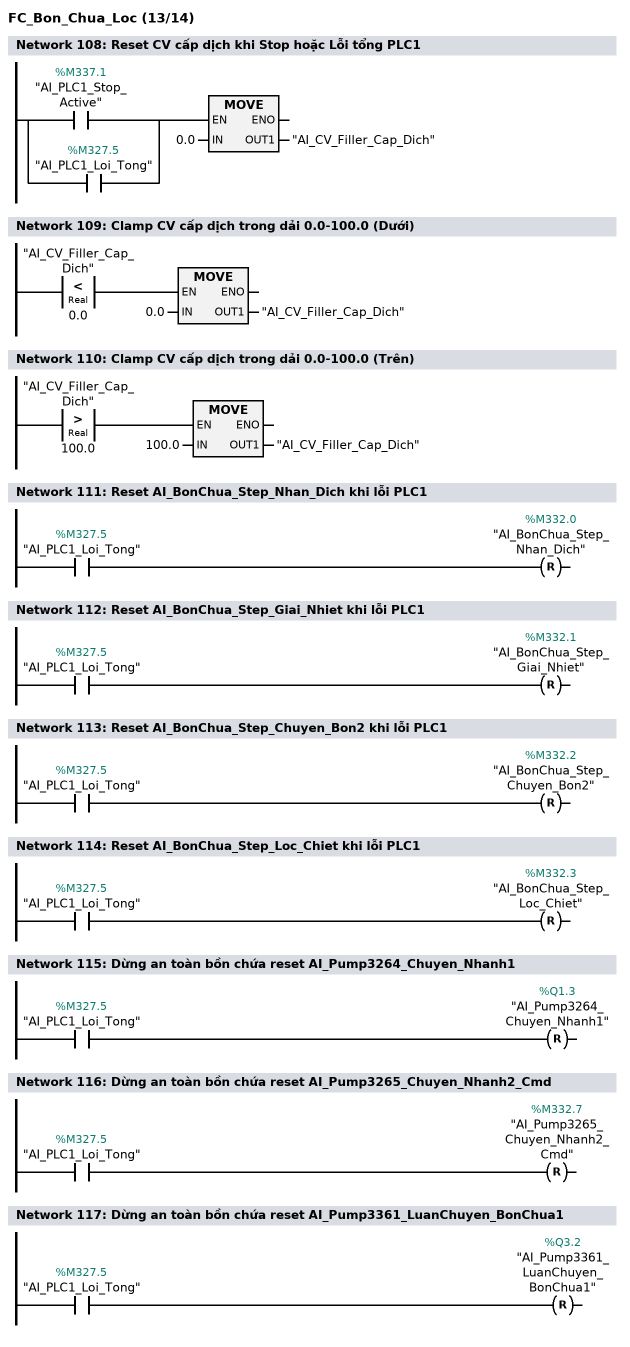
   RUNG wire#powerrail
      Contact( "AI_PLC1_Stop_Active" )
      wire#w1
      { S7_GenerateENO := "TRUE" } Move(in := 0.0, out1 => "AI_CV_Filler_Cap_Dich")
   END_RUNG
   RUNG wire#powerrail
      Contact( "AI_PLC1_Loi_Tong" )
   END_RUNG wire#w1
   // the same network as SCL:
   IF "AI_PLC1_Stop_Active" OR "AI_PLC1_Loi_Tong" THEN "AI_CV_Filler_Cap_Dich" := 0.0; END_IF;
END_REGION

REGION Network 109: Clamp CV cấp dịch trong dải 0.0-100.0 (Dưới)
   RUNG wire#powerrail
      { S7_Templates := "SrcType := Real" } LT_Contact(in1 := "AI_CV_Filler_Cap_Dich", in2 := 0.0)
      { S7_GenerateENO := "TRUE" } Move(in := 0.0, out1 => "AI_CV_Filler_Cap_Dich")
   END_RUNG
   // the same network as SCL:
   IF "AI_CV_Filler_Cap_Dich" < 0.0 THEN "AI_CV_Filler_Cap_Dich" := 0.0; END_IF;
END_REGION

REGION Network 110: Clamp CV cấp dịch trong dải 0.0-100.0 (Trên)
   RUNG wire#powerrail
      { S7_Templates := "SrcType := Real" } GT_Contact(in1 := "AI_CV_Filler_Cap_Dich", in2 := 100.0)
      { S7_GenerateENO := "TRUE" } Move(in := 100.0, out1 => "AI_CV_Filler_Cap_Dich")
   END_RUNG
   // the same network as SCL:
   IF "AI_CV_Filler_Cap_Dich" > 100.0 THEN "AI_CV_Filler_Cap_Dich" := 100.0; END_IF;
END_REGION

REGION Network 111: Reset AI_BonChua_Step_Nhan_Dich khi lỗi PLC1
   RUNG wire#powerrail
      Contact( "AI_PLC1_Loi_Tong" )
      R_Coil( "AI_BonChua_Step_Nhan_Dich" )
   END_RUNG
   // the same network as SCL:
   IF "AI_PLC1_Loi_Tong" THEN "AI_BonChua_Step_Nhan_Dich" := FALSE; END_IF;
END_REGION

REGION Network 112: Reset AI_BonChua_Step_Giai_Nhiet khi lỗi PLC1
   RUNG wire#powerrail
      Contact( "AI_PLC1_Loi_Tong" )
      R_Coil( "AI_BonChua_Step_Giai_Nhiet" )
   END_RUNG
   // the same network as SCL:
   IF "AI_PLC1_Loi_Tong" THEN "AI_BonChua_Step_Giai_Nhiet" := FALSE; END_IF;
END_REGION

REGION Network 113: Reset AI_BonChua_Step_Chuyen_Bon2 khi lỗi PLC1
   RUNG wire#powerrail
      Contact( "AI_PLC1_Loi_Tong" )
      R_Coil( "AI_BonChua_Step_Chuyen_Bon2" )
   END_RUNG
   // the same network as SCL:
   IF "AI_PLC1_Loi_Tong" THEN "AI_BonChua_Step_Chuyen_Bon2" := FALSE; END_IF;
END_REGION

REGION Network 114: Reset AI_BonChua_Step_Loc_Chiet khi lỗi PLC1
   RUNG wire#powerrail
      Contact( "AI_PLC1_Loi_Tong" )
      R_Coil( "AI_BonChua_Step_Loc_Chiet" )
   END_RUNG
   // the same network as SCL:
   IF "AI_PLC1_Loi_Tong" THEN "AI_BonChua_Step_Loc_Chiet" := FALSE; END_IF;
END_REGION

REGION Network 115: Dừng an toàn bồn chứa reset AI_Pump3264_Chuyen_Nhanh1
   RUNG wire#powerrail
      Contact( "AI_PLC1_Loi_Tong" )
      R_Coil( "AI_Pump3264_Chuyen_Nhanh1" )
   END_RUNG
   // the same network as SCL:
   IF "AI_PLC1_Loi_Tong" THEN "AI_Pump3264_Chuyen_Nhanh1" := FALSE; END_IF;
END_REGION

REGION Network 116: Dừng an toàn bồn chứa reset AI_Pump3265_Chuyen_Nhanh2_Cmd
   RUNG wire#powerrail
      Contact( "AI_PLC1_Loi_Tong" )
      R_Coil( "AI_Pump3265_Chuyen_Nhanh2_Cmd" )
   END_RUNG
   // the same network as SCL:
   IF "AI_PLC1_Loi_Tong" THEN "AI_Pump3265_Chuyen_Nhanh2_Cmd" := FALSE; END_IF;
END_REGION

REGION Network 117: Dừng an toàn bồn chứa reset AI_Pump3361_LuanChuyen_BonChua1
   RUNG wire#powerrail
      Contact( "AI_PLC1_Loi_Tong" )
      R_Coil( "AI_Pump3361_LuanChuyen_BonChua1" )
   END_RUNG
   // the same network as SCL:
   IF "AI_PLC1_Loi_Tong" THEN "AI_Pump3361_LuanChuyen_BonChua1" := FALSE; END_IF;
END_REGION

REGION Network 118: Dừng an toàn bồn chứa reset AI_Pump3362_Xa_BonChua1
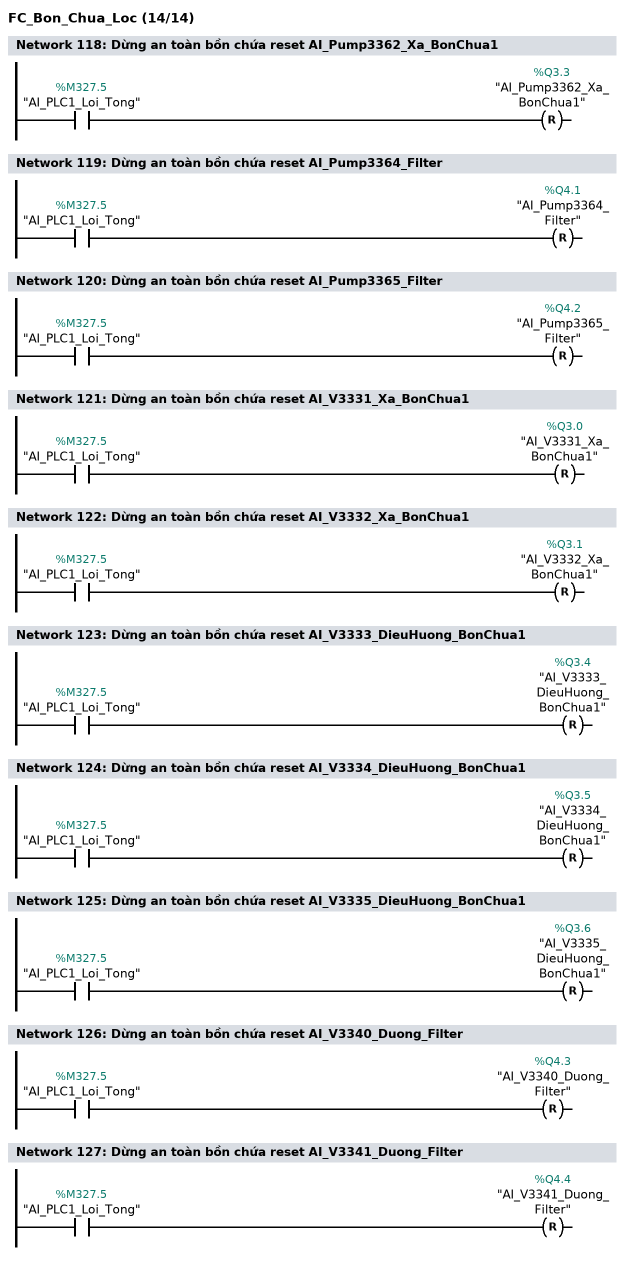
   RUNG wire#powerrail
      Contact( "AI_PLC1_Loi_Tong" )
      R_Coil( "AI_Pump3362_Xa_BonChua1" )
   END_RUNG
   // the same network as SCL:
   IF "AI_PLC1_Loi_Tong" THEN "AI_Pump3362_Xa_BonChua1" := FALSE; END_IF;
END_REGION

REGION Network 119: Dừng an toàn bồn chứa reset AI_Pump3364_Filter
   RUNG wire#powerrail
      Contact( "AI_PLC1_Loi_Tong" )
      R_Coil( "AI_Pump3364_Filter" )
   END_RUNG
   // the same network as SCL:
   IF "AI_PLC1_Loi_Tong" THEN "AI_Pump3364_Filter" := FALSE; END_IF;
END_REGION

REGION Network 120: Dừng an toàn bồn chứa reset AI_Pump3365_Filter
   RUNG wire#powerrail
      Contact( "AI_PLC1_Loi_Tong" )
      R_Coil( "AI_Pump3365_Filter" )
   END_RUNG
   // the same network as SCL:
   IF "AI_PLC1_Loi_Tong" THEN "AI_Pump3365_Filter" := FALSE; END_IF;
END_REGION

REGION Network 121: Dừng an toàn bồn chứa reset AI_V3331_Xa_BonChua1
   RUNG wire#powerrail
      Contact( "AI_PLC1_Loi_Tong" )
      R_Coil( "AI_V3331_Xa_BonChua1" )
   END_RUNG
   // the same network as SCL:
   IF "AI_PLC1_Loi_Tong" THEN "AI_V3331_Xa_BonChua1" := FALSE; END_IF;
END_REGION

REGION Network 122: Dừng an toàn bồn chứa reset AI_V3332_Xa_BonChua1
   RUNG wire#powerrail
      Contact( "AI_PLC1_Loi_Tong" )
      R_Coil( "AI_V3332_Xa_BonChua1" )
   END_RUNG
   // the same network as SCL:
   IF "AI_PLC1_Loi_Tong" THEN "AI_V3332_Xa_BonChua1" := FALSE; END_IF;
END_REGION

REGION Network 123: Dừng an toàn bồn chứa reset AI_V3333_DieuHuong_BonChua1
   RUNG wire#powerrail
      Contact( "AI_PLC1_Loi_Tong" )
      R_Coil( "AI_V3333_DieuHuong_BonChua1" )
   END_RUNG
   // the same network as SCL:
   IF "AI_PLC1_Loi_Tong" THEN "AI_V3333_DieuHuong_BonChua1" := FALSE; END_IF;
END_REGION

REGION Network 124: Dừng an toàn bồn chứa reset AI_V3334_DieuHuong_BonChua1
   RUNG wire#powerrail
      Contact( "AI_PLC1_Loi_Tong" )
      R_Coil( "AI_V3334_DieuHuong_BonChua1" )
   END_RUNG
   // the same network as SCL:
   IF "AI_PLC1_Loi_Tong" THEN "AI_V3334_DieuHuong_BonChua1" := FALSE; END_IF;
END_REGION

REGION Network 125: Dừng an toàn bồn chứa reset AI_V3335_DieuHuong_BonChua1
   RUNG wire#powerrail
      Contact( "AI_PLC1_Loi_Tong" )
      R_Coil( "AI_V3335_DieuHuong_BonChua1" )
   END_RUNG
   // the same network as SCL:
   IF "AI_PLC1_Loi_Tong" THEN "AI_V3335_DieuHuong_BonChua1" := FALSE; END_IF;
END_REGION

REGION Network 126: Dừng an toàn bồn chứa reset AI_V3340_Duong_Filter
   RUNG wire#powerrail
      Contact( "AI_PLC1_Loi_Tong" )
      R_Coil( "AI_V3340_Duong_Filter" )
   END_RUNG
   // the same network as SCL:
   IF "AI_PLC1_Loi_Tong" THEN "AI_V3340_Duong_Filter" := FALSE; END_IF;
END_REGION

REGION Network 127: Dừng an toàn bồn chứa reset AI_V3341_Duong_Filter
   RUNG wire#powerrail
      Contact( "AI_PLC1_Loi_Tong" )
      R_Coil( "AI_V3341_Duong_Filter" )
   END_RUNG
   // the same network as SCL:
   IF "AI_PLC1_Loi_Tong" THEN "AI_V3341_Duong_Filter" := FALSE; END_IF;
END_REGION
END_FUNCTION

FUNCTION "FC_HMI_Mirror_PLC1" : Void   // FC40, LAD
{ S7_Optimized_Access := 'TRUE' }
VERSION : 0.1
// stored: AutoNumber true, IsIECCheckEnabled false, SetENOAutomatically false, UDAEnableTagReadback false
BEGIN

REGION Network 1: Mirror AI_V3230_Nuoc_Bon1
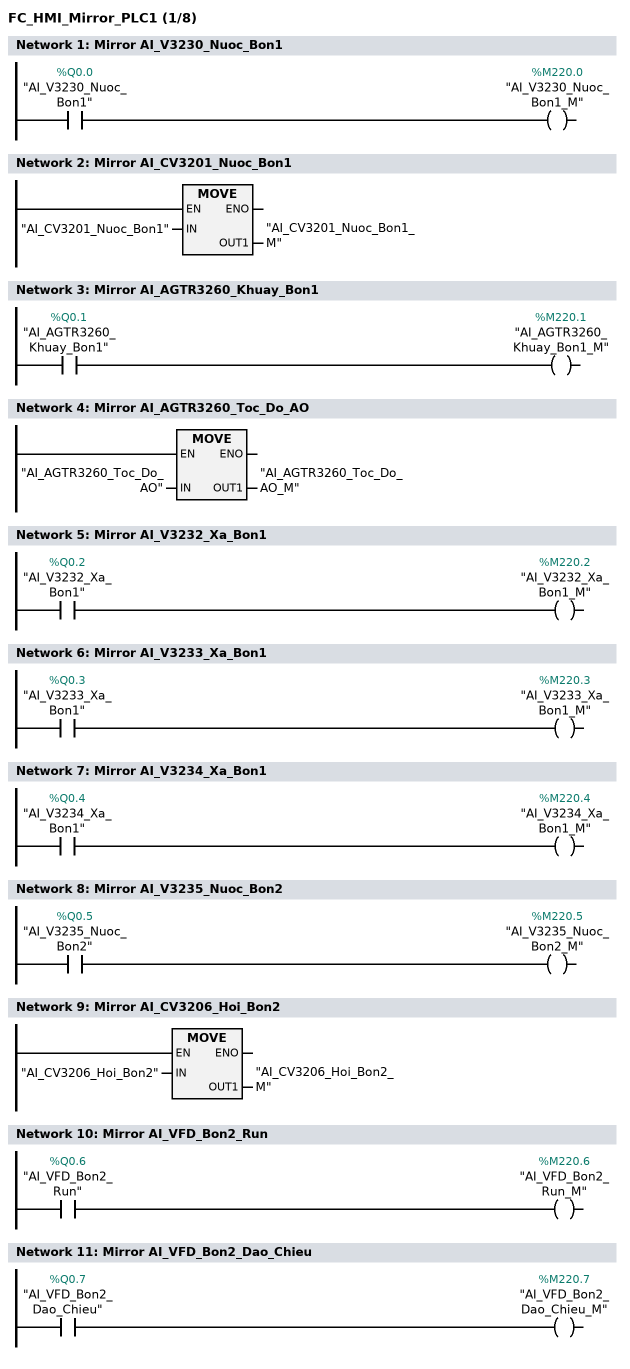
   RUNG wire#powerrail
      Contact( "AI_V3230_Nuoc_Bon1" )
      Coil( "AI_V3230_Nuoc_Bon1_M" )
   END_RUNG
   // the same network as SCL:
   "AI_V3230_Nuoc_Bon1_M" := "AI_V3230_Nuoc_Bon1";
END_REGION

REGION Network 2: Mirror AI_CV3201_Nuoc_Bon1
   RUNG wire#powerrail
      { S7_GenerateENO := "TRUE" } Move(in := "AI_CV3201_Nuoc_Bon1", out1 => "AI_CV3201_Nuoc_Bon1_M")
   END_RUNG
   // the same network as SCL:
   "AI_CV3201_Nuoc_Bon1_M" := "AI_CV3201_Nuoc_Bon1";
END_REGION

REGION Network 3: Mirror AI_AGTR3260_Khuay_Bon1
   RUNG wire#powerrail
      Contact( "AI_AGTR3260_Khuay_Bon1" )
      Coil( "AI_AGTR3260_Khuay_Bon1_M" )
   END_RUNG
   // the same network as SCL:
   "AI_AGTR3260_Khuay_Bon1_M" := "AI_AGTR3260_Khuay_Bon1";
END_REGION

REGION Network 4: Mirror AI_AGTR3260_Toc_Do_AO
   RUNG wire#powerrail
      { S7_GenerateENO := "TRUE" } Move(in := "AI_AGTR3260_Toc_Do_AO", out1 => "AI_AGTR3260_Toc_Do_AO_M")
   END_RUNG
   // the same network as SCL:
   "AI_AGTR3260_Toc_Do_AO_M" := "AI_AGTR3260_Toc_Do_AO";
END_REGION

REGION Network 5: Mirror AI_V3232_Xa_Bon1
   RUNG wire#powerrail
      Contact( "AI_V3232_Xa_Bon1" )
      Coil( "AI_V3232_Xa_Bon1_M" )
   END_RUNG
   // the same network as SCL:
   "AI_V3232_Xa_Bon1_M" := "AI_V3232_Xa_Bon1";
END_REGION

REGION Network 6: Mirror AI_V3233_Xa_Bon1
   RUNG wire#powerrail
      Contact( "AI_V3233_Xa_Bon1" )
      Coil( "AI_V3233_Xa_Bon1_M" )
   END_RUNG
   // the same network as SCL:
   "AI_V3233_Xa_Bon1_M" := "AI_V3233_Xa_Bon1";
END_REGION

REGION Network 7: Mirror AI_V3234_Xa_Bon1
   RUNG wire#powerrail
      Contact( "AI_V3234_Xa_Bon1" )
      Coil( "AI_V3234_Xa_Bon1_M" )
   END_RUNG
   // the same network as SCL:
   "AI_V3234_Xa_Bon1_M" := "AI_V3234_Xa_Bon1";
END_REGION

REGION Network 8: Mirror AI_V3235_Nuoc_Bon2
   RUNG wire#powerrail
      Contact( "AI_V3235_Nuoc_Bon2" )
      Coil( "AI_V3235_Nuoc_Bon2_M" )
   END_RUNG
   // the same network as SCL:
   "AI_V3235_Nuoc_Bon2_M" := "AI_V3235_Nuoc_Bon2";
END_REGION

REGION Network 9: Mirror AI_CV3206_Hoi_Bon2
   RUNG wire#powerrail
      { S7_GenerateENO := "TRUE" } Move(in := "AI_CV3206_Hoi_Bon2", out1 => "AI_CV3206_Hoi_Bon2_M")
   END_RUNG
   // the same network as SCL:
   "AI_CV3206_Hoi_Bon2_M" := "AI_CV3206_Hoi_Bon2";
END_REGION

REGION Network 10: Mirror AI_VFD_Bon2_Run
   RUNG wire#powerrail
      Contact( "AI_VFD_Bon2_Run" )
      Coil( "AI_VFD_Bon2_Run_M" )
   END_RUNG
   // the same network as SCL:
   "AI_VFD_Bon2_Run_M" := "AI_VFD_Bon2_Run";
END_REGION

REGION Network 11: Mirror AI_VFD_Bon2_Dao_Chieu
   RUNG wire#powerrail
      Contact( "AI_VFD_Bon2_Dao_Chieu" )
      Coil( "AI_VFD_Bon2_Dao_Chieu_M" )
   END_RUNG
   // the same network as SCL:
   "AI_VFD_Bon2_Dao_Chieu_M" := "AI_VFD_Bon2_Dao_Chieu";
END_REGION

REGION Network 12: Mirror AI_VFD_Bon2_Toc_Do_AO
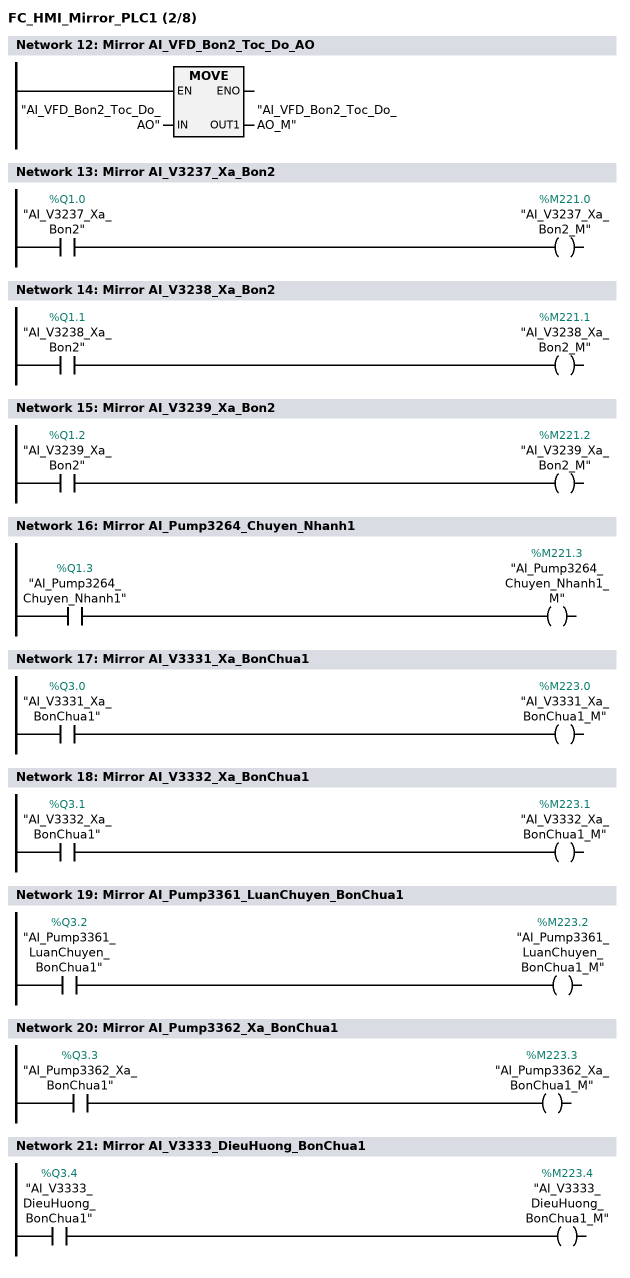
   RUNG wire#powerrail
      { S7_GenerateENO := "TRUE" } Move(in := "AI_VFD_Bon2_Toc_Do_AO", out1 => "AI_VFD_Bon2_Toc_Do_AO_M")
   END_RUNG
   // the same network as SCL:
   "AI_VFD_Bon2_Toc_Do_AO_M" := "AI_VFD_Bon2_Toc_Do_AO";
END_REGION

REGION Network 13: Mirror AI_V3237_Xa_Bon2
   RUNG wire#powerrail
      Contact( "AI_V3237_Xa_Bon2" )
      Coil( "AI_V3237_Xa_Bon2_M" )
   END_RUNG
   // the same network as SCL:
   "AI_V3237_Xa_Bon2_M" := "AI_V3237_Xa_Bon2";
END_REGION

REGION Network 14: Mirror AI_V3238_Xa_Bon2
   RUNG wire#powerrail
      Contact( "AI_V3238_Xa_Bon2" )
      Coil( "AI_V3238_Xa_Bon2_M" )
   END_RUNG
   // the same network as SCL:
   "AI_V3238_Xa_Bon2_M" := "AI_V3238_Xa_Bon2";
END_REGION

REGION Network 15: Mirror AI_V3239_Xa_Bon2
   RUNG wire#powerrail
      Contact( "AI_V3239_Xa_Bon2" )
      Coil( "AI_V3239_Xa_Bon2_M" )
   END_RUNG
   // the same network as SCL:
   "AI_V3239_Xa_Bon2_M" := "AI_V3239_Xa_Bon2";
END_REGION

REGION Network 16: Mirror AI_Pump3264_Chuyen_Nhanh1
   RUNG wire#powerrail
      Contact( "AI_Pump3264_Chuyen_Nhanh1" )
      Coil( "AI_Pump3264_Chuyen_Nhanh1_M" )
   END_RUNG
   // the same network as SCL:
   "AI_Pump3264_Chuyen_Nhanh1_M" := "AI_Pump3264_Chuyen_Nhanh1";
END_REGION

REGION Network 17: Mirror AI_V3331_Xa_BonChua1
   RUNG wire#powerrail
      Contact( "AI_V3331_Xa_BonChua1" )
      Coil( "AI_V3331_Xa_BonChua1_M" )
   END_RUNG
   // the same network as SCL:
   "AI_V3331_Xa_BonChua1_M" := "AI_V3331_Xa_BonChua1";
END_REGION

REGION Network 18: Mirror AI_V3332_Xa_BonChua1
   RUNG wire#powerrail
      Contact( "AI_V3332_Xa_BonChua1" )
      Coil( "AI_V3332_Xa_BonChua1_M" )
   END_RUNG
   // the same network as SCL:
   "AI_V3332_Xa_BonChua1_M" := "AI_V3332_Xa_BonChua1";
END_REGION

REGION Network 19: Mirror AI_Pump3361_LuanChuyen_BonChua1
   RUNG wire#powerrail
      Contact( "AI_Pump3361_LuanChuyen_BonChua1" )
      Coil( "AI_Pump3361_LuanChuyen_BonChua1_M" )
   END_RUNG
   // the same network as SCL:
   "AI_Pump3361_LuanChuyen_BonChua1_M" := "AI_Pump3361_LuanChuyen_BonChua1";
END_REGION

REGION Network 20: Mirror AI_Pump3362_Xa_BonChua1
   RUNG wire#powerrail
      Contact( "AI_Pump3362_Xa_BonChua1" )
      Coil( "AI_Pump3362_Xa_BonChua1_M" )
   END_RUNG
   // the same network as SCL:
   "AI_Pump3362_Xa_BonChua1_M" := "AI_Pump3362_Xa_BonChua1";
END_REGION

REGION Network 21: Mirror AI_V3333_DieuHuong_BonChua1
   RUNG wire#powerrail
      Contact( "AI_V3333_DieuHuong_BonChua1" )
      Coil( "AI_V3333_DieuHuong_BonChua1_M" )
   END_RUNG
   // the same network as SCL:
   "AI_V3333_DieuHuong_BonChua1_M" := "AI_V3333_DieuHuong_BonChua1";
END_REGION

REGION Network 22: Mirror AI_V3334_DieuHuong_BonChua1
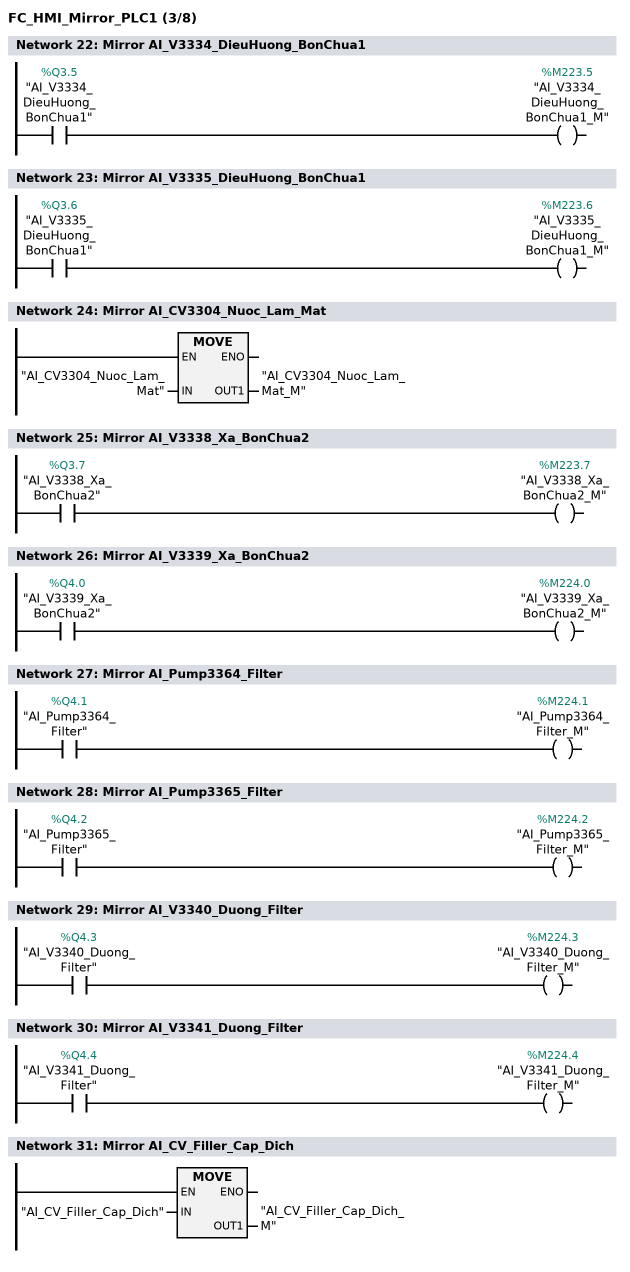
   RUNG wire#powerrail
      Contact( "AI_V3334_DieuHuong_BonChua1" )
      Coil( "AI_V3334_DieuHuong_BonChua1_M" )
   END_RUNG
   // the same network as SCL:
   "AI_V3334_DieuHuong_BonChua1_M" := "AI_V3334_DieuHuong_BonChua1";
END_REGION

REGION Network 23: Mirror AI_V3335_DieuHuong_BonChua1
   RUNG wire#powerrail
      Contact( "AI_V3335_DieuHuong_BonChua1" )
      Coil( "AI_V3335_DieuHuong_BonChua1_M" )
   END_RUNG
   // the same network as SCL:
   "AI_V3335_DieuHuong_BonChua1_M" := "AI_V3335_DieuHuong_BonChua1";
END_REGION

REGION Network 24: Mirror AI_CV3304_Nuoc_Lam_Mat
   RUNG wire#powerrail
      { S7_GenerateENO := "TRUE" } Move(in := "AI_CV3304_Nuoc_Lam_Mat", out1 => "AI_CV3304_Nuoc_Lam_Mat_M")
   END_RUNG
   // the same network as SCL:
   "AI_CV3304_Nuoc_Lam_Mat_M" := "AI_CV3304_Nuoc_Lam_Mat";
END_REGION

REGION Network 25: Mirror AI_V3338_Xa_BonChua2
   RUNG wire#powerrail
      Contact( "AI_V3338_Xa_BonChua2" )
      Coil( "AI_V3338_Xa_BonChua2_M" )
   END_RUNG
   // the same network as SCL:
   "AI_V3338_Xa_BonChua2_M" := "AI_V3338_Xa_BonChua2";
END_REGION

REGION Network 26: Mirror AI_V3339_Xa_BonChua2
   RUNG wire#powerrail
      Contact( "AI_V3339_Xa_BonChua2" )
      Coil( "AI_V3339_Xa_BonChua2_M" )
   END_RUNG
   // the same network as SCL:
   "AI_V3339_Xa_BonChua2_M" := "AI_V3339_Xa_BonChua2";
END_REGION

REGION Network 27: Mirror AI_Pump3364_Filter
   RUNG wire#powerrail
      Contact( "AI_Pump3364_Filter" )
      Coil( "AI_Pump3364_Filter_M" )
   END_RUNG
   // the same network as SCL:
   "AI_Pump3364_Filter_M" := "AI_Pump3364_Filter";
END_REGION

REGION Network 28: Mirror AI_Pump3365_Filter
   RUNG wire#powerrail
      Contact( "AI_Pump3365_Filter" )
      Coil( "AI_Pump3365_Filter_M" )
   END_RUNG
   // the same network as SCL:
   "AI_Pump3365_Filter_M" := "AI_Pump3365_Filter";
END_REGION

REGION Network 29: Mirror AI_V3340_Duong_Filter
   RUNG wire#powerrail
      Contact( "AI_V3340_Duong_Filter" )
      Coil( "AI_V3340_Duong_Filter_M" )
   END_RUNG
   // the same network as SCL:
   "AI_V3340_Duong_Filter_M" := "AI_V3340_Duong_Filter";
END_REGION

REGION Network 30: Mirror AI_V3341_Duong_Filter
   RUNG wire#powerrail
      Contact( "AI_V3341_Duong_Filter" )
      Coil( "AI_V3341_Duong_Filter_M" )
   END_RUNG
   // the same network as SCL:
   "AI_V3341_Duong_Filter_M" := "AI_V3341_Duong_Filter";
END_REGION

REGION Network 31: Mirror AI_CV_Filler_Cap_Dich
   RUNG wire#powerrail
      { S7_GenerateENO := "TRUE" } Move(in := "AI_CV_Filler_Cap_Dich", out1 => "AI_CV_Filler_Cap_Dich_M")
   END_RUNG
   // the same network as SCL:
   "AI_CV_Filler_Cap_Dich_M" := "AI_CV_Filler_Cap_Dich";
END_REGION

REGION Network 32: Mirror AI_Coi_Bao_Dong
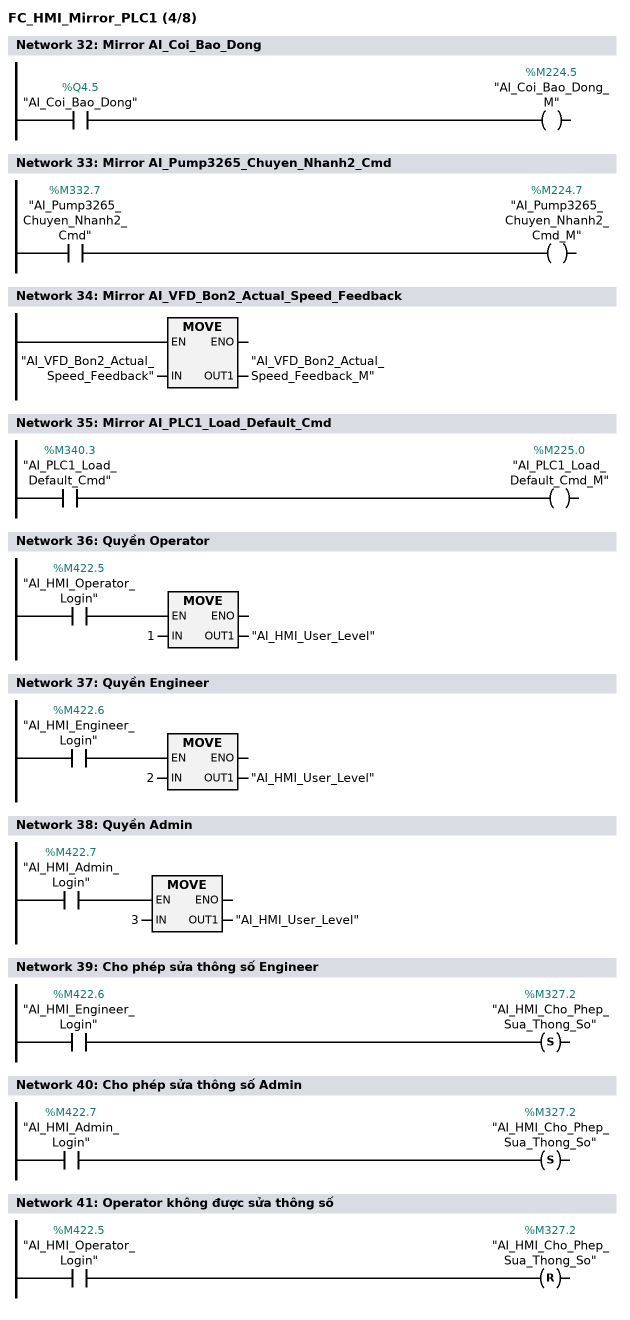
   RUNG wire#powerrail
      Contact( "AI_Coi_Bao_Dong" )
      Coil( "AI_Coi_Bao_Dong_M" )
   END_RUNG
   // the same network as SCL:
   "AI_Coi_Bao_Dong_M" := "AI_Coi_Bao_Dong";
END_REGION

REGION Network 33: Mirror AI_Pump3265_Chuyen_Nhanh2_Cmd
   RUNG wire#powerrail
      Contact( "AI_Pump3265_Chuyen_Nhanh2_Cmd" )
      Coil( "AI_Pump3265_Chuyen_Nhanh2_Cmd_M" )
   END_RUNG
   // the same network as SCL:
   "AI_Pump3265_Chuyen_Nhanh2_Cmd_M" := "AI_Pump3265_Chuyen_Nhanh2_Cmd";
END_REGION

REGION Network 34: Mirror AI_VFD_Bon2_Actual_Speed_Feedback
   RUNG wire#powerrail
      { S7_GenerateENO := "TRUE" } Move(in := "AI_VFD_Bon2_Actual_Speed_Feedback", out1 => "AI_VFD_Bon2_Actual_Speed_Feedback_M")
   END_RUNG
   // the same network as SCL:
   "AI_VFD_Bon2_Actual_Speed_Feedback_M" := "AI_VFD_Bon2_Actual_Speed_Feedback";
END_REGION

REGION Network 35: Mirror AI_PLC1_Load_Default_Cmd
   RUNG wire#powerrail
      Contact( "AI_PLC1_Load_Default_Cmd" )
      Coil( "AI_PLC1_Load_Default_Cmd_M" )
   END_RUNG
   // the same network as SCL:
   "AI_PLC1_Load_Default_Cmd_M" := "AI_PLC1_Load_Default_Cmd";
END_REGION

REGION Network 36: Quyền Operator
   RUNG wire#powerrail
      Contact( "AI_HMI_Operator_Login" )
      { S7_GenerateENO := "TRUE" } Move(in := 1, out1 => "AI_HMI_User_Level")
   END_RUNG
   // the same network as SCL:
   IF "AI_HMI_Operator_Login" THEN "AI_HMI_User_Level" := 1; END_IF;
END_REGION

REGION Network 37: Quyền Engineer
   RUNG wire#powerrail
      Contact( "AI_HMI_Engineer_Login" )
      { S7_GenerateENO := "TRUE" } Move(in := 2, out1 => "AI_HMI_User_Level")
   END_RUNG
   // the same network as SCL:
   IF "AI_HMI_Engineer_Login" THEN "AI_HMI_User_Level" := 2; END_IF;
END_REGION

REGION Network 38: Quyền Admin
   RUNG wire#powerrail
      Contact( "AI_HMI_Admin_Login" )
      { S7_GenerateENO := "TRUE" } Move(in := 3, out1 => "AI_HMI_User_Level")
   END_RUNG
   // the same network as SCL:
   IF "AI_HMI_Admin_Login" THEN "AI_HMI_User_Level" := 3; END_IF;
END_REGION

REGION Network 39: Cho phép sửa thông số Engineer
   RUNG wire#powerrail
      Contact( "AI_HMI_Engineer_Login" )
      S_Coil( "AI_HMI_Cho_Phep_Sua_Thong_So" )
   END_RUNG
   // the same network as SCL:
   IF "AI_HMI_Engineer_Login" THEN "AI_HMI_Cho_Phep_Sua_Thong_So" := TRUE; END_IF;
END_REGION

REGION Network 40: Cho phép sửa thông số Admin
   RUNG wire#powerrail
      Contact( "AI_HMI_Admin_Login" )
      S_Coil( "AI_HMI_Cho_Phep_Sua_Thong_So" )
   END_RUNG
   // the same network as SCL:
   IF "AI_HMI_Admin_Login" THEN "AI_HMI_Cho_Phep_Sua_Thong_So" := TRUE; END_IF;
END_REGION

REGION Network 41: Operator không được sửa thông số
   RUNG wire#powerrail
      Contact( "AI_HMI_Operator_Login" )
      R_Coil( "AI_HMI_Cho_Phep_Sua_Thong_So" )
   END_RUNG
   // the same network as SCL:
   IF "AI_HMI_Operator_Login" THEN "AI_HMI_Cho_Phep_Sua_Thong_So" := FALSE; END_IF;
END_REGION

REGION Network 42: Mã an toàn mặc định
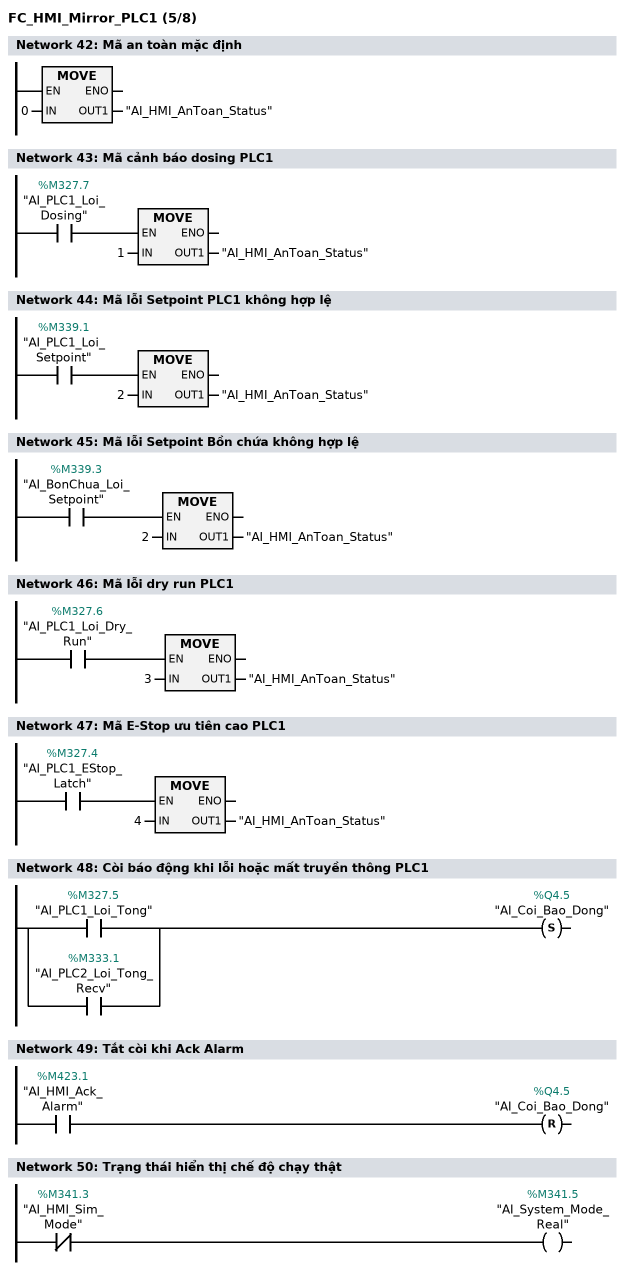
   RUNG wire#powerrail
      { S7_GenerateENO := "TRUE" } Move(in := 0, out1 => "AI_HMI_AnToan_Status")
   END_RUNG
   // the same network as SCL:
   "AI_HMI_AnToan_Status" := 0;
END_REGION

REGION Network 43: Mã cảnh báo dosing PLC1
   RUNG wire#powerrail
      Contact( "AI_PLC1_Loi_Dosing" )
      { S7_GenerateENO := "TRUE" } Move(in := 1, out1 => "AI_HMI_AnToan_Status")
   END_RUNG
   // the same network as SCL:
   IF "AI_PLC1_Loi_Dosing" THEN "AI_HMI_AnToan_Status" := 1; END_IF;
END_REGION

REGION Network 44: Mã lỗi Setpoint PLC1 không hợp lệ
   RUNG wire#powerrail
      Contact( "AI_PLC1_Loi_Setpoint" )
      { S7_GenerateENO := "TRUE" } Move(in := 2, out1 => "AI_HMI_AnToan_Status")
   END_RUNG
   // the same network as SCL:
   IF "AI_PLC1_Loi_Setpoint" THEN "AI_HMI_AnToan_Status" := 2; END_IF;
END_REGION

REGION Network 45: Mã lỗi Setpoint Bồn chứa không hợp lệ
   RUNG wire#powerrail
      Contact( "AI_BonChua_Loi_Setpoint" )
      { S7_GenerateENO := "TRUE" } Move(in := 2, out1 => "AI_HMI_AnToan_Status")
   END_RUNG
   // the same network as SCL:
   IF "AI_BonChua_Loi_Setpoint" THEN "AI_HMI_AnToan_Status" := 2; END_IF;
END_REGION

REGION Network 46: Mã lỗi dry run PLC1
   RUNG wire#powerrail
      Contact( "AI_PLC1_Loi_Dry_Run" )
      { S7_GenerateENO := "TRUE" } Move(in := 3, out1 => "AI_HMI_AnToan_Status")
   END_RUNG
   // the same network as SCL:
   IF "AI_PLC1_Loi_Dry_Run" THEN "AI_HMI_AnToan_Status" := 3; END_IF;
END_REGION

REGION Network 47: Mã E-Stop ưu tiên cao PLC1
   RUNG wire#powerrail
      Contact( "AI_PLC1_EStop_Latch" )
      { S7_GenerateENO := "TRUE" } Move(in := 4, out1 => "AI_HMI_AnToan_Status")
   END_RUNG
   // the same network as SCL:
   IF "AI_PLC1_EStop_Latch" THEN "AI_HMI_AnToan_Status" := 4; END_IF;
END_REGION

REGION Network 48: Còi báo động khi lỗi hoặc mất truyền thông PLC1
   RUNG wire#powerrail
      Contact( "AI_PLC1_Loi_Tong" )
      wire#w1
      S_Coil( "AI_Coi_Bao_Dong" )
   END_RUNG
   RUNG wire#powerrail
      Contact( "AI_PLC2_Loi_Tong_Recv" )
   END_RUNG wire#w1
   // the same network as SCL:
   IF "AI_PLC1_Loi_Tong" OR "AI_PLC2_Loi_Tong_Recv" THEN "AI_Coi_Bao_Dong" := TRUE; END_IF;
END_REGION

REGION Network 49: Tắt còi khi Ack Alarm
   RUNG wire#powerrail
      Contact( "AI_HMI_Ack_Alarm" )
      R_Coil( "AI_Coi_Bao_Dong" )
   END_RUNG
   // the same network as SCL:
   IF "AI_HMI_Ack_Alarm" THEN "AI_Coi_Bao_Dong" := FALSE; END_IF;
END_REGION

REGION Network 50: Trạng thái hiển thị chế độ chạy thật
   RUNG wire#powerrail
      I_Contact( "AI_HMI_Sim_Mode" )
      Coil( "AI_System_Mode_Real" )
   END_RUNG
   // the same network as SCL:
   "AI_System_Mode_Real" := NOT "AI_HMI_Sim_Mode";
END_REGION

REGION Network 51: Trạng thái hiển thị chế độ mô phỏng
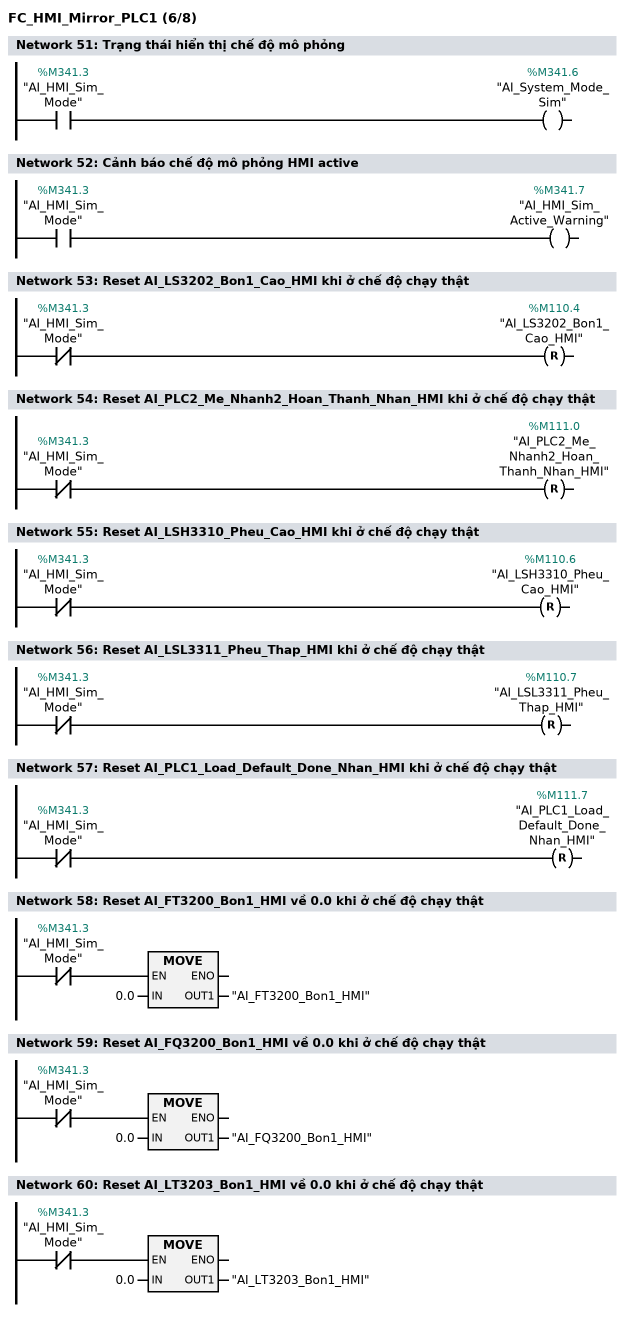
   RUNG wire#powerrail
      Contact( "AI_HMI_Sim_Mode" )
      Coil( "AI_System_Mode_Sim" )
   END_RUNG
   // the same network as SCL:
   "AI_System_Mode_Sim" := "AI_HMI_Sim_Mode";
END_REGION

REGION Network 52: Cảnh báo chế độ mô phỏng HMI active
   RUNG wire#powerrail
      Contact( "AI_HMI_Sim_Mode" )
      Coil( "AI_HMI_Sim_Active_Warning" )
   END_RUNG
   // the same network as SCL:
   "AI_HMI_Sim_Active_Warning" := "AI_HMI_Sim_Mode";
END_REGION

REGION Network 53: Reset AI_LS3202_Bon1_Cao_HMI khi ở chế độ chạy thật
   RUNG wire#powerrail
      I_Contact( "AI_HMI_Sim_Mode" )
      R_Coil( "AI_LS3202_Bon1_Cao_HMI" )
   END_RUNG
   // the same network as SCL:
   IF NOT "AI_HMI_Sim_Mode" THEN "AI_LS3202_Bon1_Cao_HMI" := FALSE; END_IF;
END_REGION

REGION Network 54: Reset AI_PLC2_Me_Nhanh2_Hoan_Thanh_Nhan_HMI khi ở chế độ chạy thật
   RUNG wire#powerrail
      I_Contact( "AI_HMI_Sim_Mode" )
      R_Coil( "AI_PLC2_Me_Nhanh2_Hoan_Thanh_Nhan_HMI" )
   END_RUNG
   // the same network as SCL:
   IF NOT "AI_HMI_Sim_Mode" THEN "AI_PLC2_Me_Nhanh2_Hoan_Thanh_Nhan_HMI" := FALSE; END_IF;
END_REGION

REGION Network 55: Reset AI_LSH3310_Pheu_Cao_HMI khi ở chế độ chạy thật
   RUNG wire#powerrail
      I_Contact( "AI_HMI_Sim_Mode" )
      R_Coil( "AI_LSH3310_Pheu_Cao_HMI" )
   END_RUNG
   // the same network as SCL:
   IF NOT "AI_HMI_Sim_Mode" THEN "AI_LSH3310_Pheu_Cao_HMI" := FALSE; END_IF;
END_REGION

REGION Network 56: Reset AI_LSL3311_Pheu_Thap_HMI khi ở chế độ chạy thật
   RUNG wire#powerrail
      I_Contact( "AI_HMI_Sim_Mode" )
      R_Coil( "AI_LSL3311_Pheu_Thap_HMI" )
   END_RUNG
   // the same network as SCL:
   IF NOT "AI_HMI_Sim_Mode" THEN "AI_LSL3311_Pheu_Thap_HMI" := FALSE; END_IF;
END_REGION

REGION Network 57: Reset AI_PLC1_Load_Default_Done_Nhan_HMI khi ở chế độ chạy thật
   RUNG wire#powerrail
      I_Contact( "AI_HMI_Sim_Mode" )
      R_Coil( "AI_PLC1_Load_Default_Done_Nhan_HMI" )
   END_RUNG
   // the same network as SCL:
   IF NOT "AI_HMI_Sim_Mode" THEN "AI_PLC1_Load_Default_Done_Nhan_HMI" := FALSE; END_IF;
END_REGION

REGION Network 58: Reset AI_FT3200_Bon1_HMI về 0.0 khi ở chế độ chạy thật
   RUNG wire#powerrail
      I_Contact( "AI_HMI_Sim_Mode" )
      { S7_GenerateENO := "TRUE" } Move(in := 0.0, out1 => "AI_FT3200_Bon1_HMI")
   END_RUNG
   // the same network as SCL:
   IF NOT "AI_HMI_Sim_Mode" THEN "AI_FT3200_Bon1_HMI" := 0.0; END_IF;
END_REGION

REGION Network 59: Reset AI_FQ3200_Bon1_HMI về 0.0 khi ở chế độ chạy thật
   RUNG wire#powerrail
      I_Contact( "AI_HMI_Sim_Mode" )
      { S7_GenerateENO := "TRUE" } Move(in := 0.0, out1 => "AI_FQ3200_Bon1_HMI")
   END_RUNG
   // the same network as SCL:
   IF NOT "AI_HMI_Sim_Mode" THEN "AI_FQ3200_Bon1_HMI" := 0.0; END_IF;
END_REGION

REGION Network 60: Reset AI_LT3203_Bon1_HMI về 0.0 khi ở chế độ chạy thật
   RUNG wire#powerrail
      I_Contact( "AI_HMI_Sim_Mode" )
      { S7_GenerateENO := "TRUE" } Move(in := 0.0, out1 => "AI_LT3203_Bon1_HMI")
   END_RUNG
   // the same network as SCL:
   IF NOT "AI_HMI_Sim_Mode" THEN "AI_LT3203_Bon1_HMI" := 0.0; END_IF;
END_REGION

REGION Network 61: Reset AI_TT3204_Bon1_HMI về 0.0 khi ở chế độ chạy thật
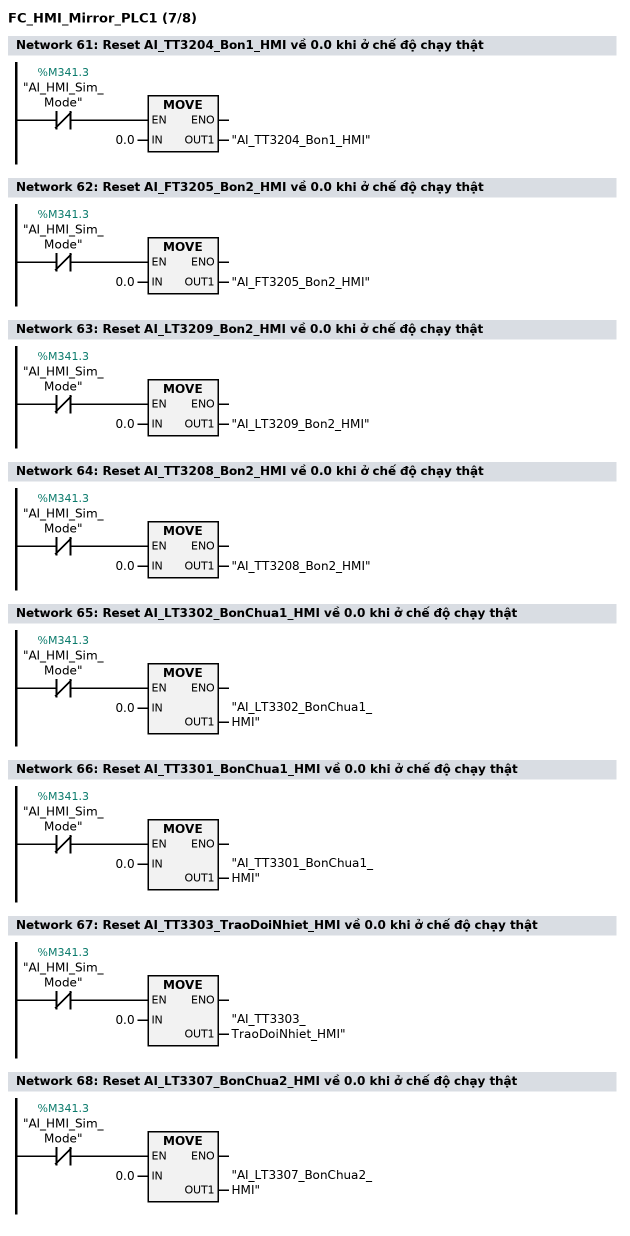
   RUNG wire#powerrail
      I_Contact( "AI_HMI_Sim_Mode" )
      { S7_GenerateENO := "TRUE" } Move(in := 0.0, out1 => "AI_TT3204_Bon1_HMI")
   END_RUNG
   // the same network as SCL:
   IF NOT "AI_HMI_Sim_Mode" THEN "AI_TT3204_Bon1_HMI" := 0.0; END_IF;
END_REGION

REGION Network 62: Reset AI_FT3205_Bon2_HMI về 0.0 khi ở chế độ chạy thật
   RUNG wire#powerrail
      I_Contact( "AI_HMI_Sim_Mode" )
      { S7_GenerateENO := "TRUE" } Move(in := 0.0, out1 => "AI_FT3205_Bon2_HMI")
   END_RUNG
   // the same network as SCL:
   IF NOT "AI_HMI_Sim_Mode" THEN "AI_FT3205_Bon2_HMI" := 0.0; END_IF;
END_REGION

REGION Network 63: Reset AI_LT3209_Bon2_HMI về 0.0 khi ở chế độ chạy thật
   RUNG wire#powerrail
      I_Contact( "AI_HMI_Sim_Mode" )
      { S7_GenerateENO := "TRUE" } Move(in := 0.0, out1 => "AI_LT3209_Bon2_HMI")
   END_RUNG
   // the same network as SCL:
   IF NOT "AI_HMI_Sim_Mode" THEN "AI_LT3209_Bon2_HMI" := 0.0; END_IF;
END_REGION

REGION Network 64: Reset AI_TT3208_Bon2_HMI về 0.0 khi ở chế độ chạy thật
   RUNG wire#powerrail
      I_Contact( "AI_HMI_Sim_Mode" )
      { S7_GenerateENO := "TRUE" } Move(in := 0.0, out1 => "AI_TT3208_Bon2_HMI")
   END_RUNG
   // the same network as SCL:
   IF NOT "AI_HMI_Sim_Mode" THEN "AI_TT3208_Bon2_HMI" := 0.0; END_IF;
END_REGION

REGION Network 65: Reset AI_LT3302_BonChua1_HMI về 0.0 khi ở chế độ chạy thật
   RUNG wire#powerrail
      I_Contact( "AI_HMI_Sim_Mode" )
      { S7_GenerateENO := "TRUE" } Move(in := 0.0, out1 => "AI_LT3302_BonChua1_HMI")
   END_RUNG
   // the same network as SCL:
   IF NOT "AI_HMI_Sim_Mode" THEN "AI_LT3302_BonChua1_HMI" := 0.0; END_IF;
END_REGION

REGION Network 66: Reset AI_TT3301_BonChua1_HMI về 0.0 khi ở chế độ chạy thật
   RUNG wire#powerrail
      I_Contact( "AI_HMI_Sim_Mode" )
      { S7_GenerateENO := "TRUE" } Move(in := 0.0, out1 => "AI_TT3301_BonChua1_HMI")
   END_RUNG
   // the same network as SCL:
   IF NOT "AI_HMI_Sim_Mode" THEN "AI_TT3301_BonChua1_HMI" := 0.0; END_IF;
END_REGION

REGION Network 67: Reset AI_TT3303_TraoDoiNhiet_HMI về 0.0 khi ở chế độ chạy thật
   RUNG wire#powerrail
      I_Contact( "AI_HMI_Sim_Mode" )
      { S7_GenerateENO := "TRUE" } Move(in := 0.0, out1 => "AI_TT3303_TraoDoiNhiet_HMI")
   END_RUNG
   // the same network as SCL:
   IF NOT "AI_HMI_Sim_Mode" THEN "AI_TT3303_TraoDoiNhiet_HMI" := 0.0; END_IF;
END_REGION

REGION Network 68: Reset AI_LT3307_BonChua2_HMI về 0.0 khi ở chế độ chạy thật
   RUNG wire#powerrail
      I_Contact( "AI_HMI_Sim_Mode" )
      { S7_GenerateENO := "TRUE" } Move(in := 0.0, out1 => "AI_LT3307_BonChua2_HMI")
   END_RUNG
   // the same network as SCL:
   IF NOT "AI_HMI_Sim_Mode" THEN "AI_LT3307_BonChua2_HMI" := 0.0; END_IF;
END_REGION

REGION Network 69: Reset AI_TT3306_BonChua2_HMI về 0.0 khi ở chế độ chạy thật
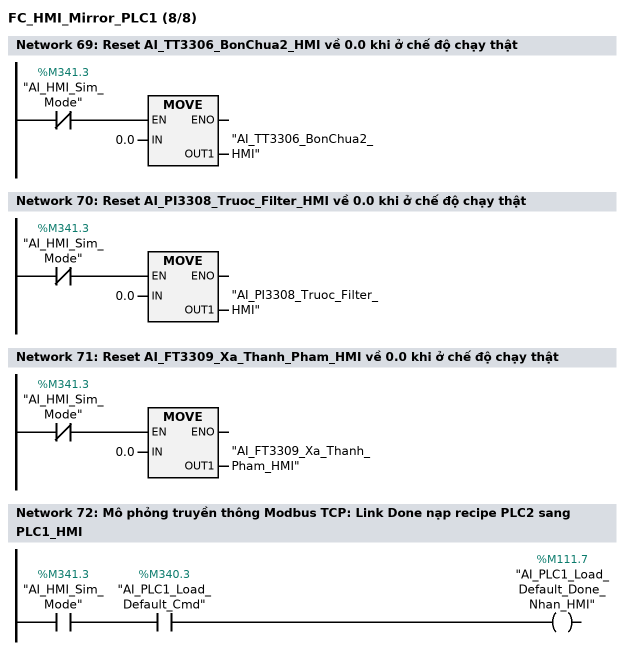
   RUNG wire#powerrail
      I_Contact( "AI_HMI_Sim_Mode" )
      { S7_GenerateENO := "TRUE" } Move(in := 0.0, out1 => "AI_TT3306_BonChua2_HMI")
   END_RUNG
   // the same network as SCL:
   IF NOT "AI_HMI_Sim_Mode" THEN "AI_TT3306_BonChua2_HMI" := 0.0; END_IF;
END_REGION

REGION Network 70: Reset AI_PI3308_Truoc_Filter_HMI về 0.0 khi ở chế độ chạy thật
   RUNG wire#powerrail
      I_Contact( "AI_HMI_Sim_Mode" )
      { S7_GenerateENO := "TRUE" } Move(in := 0.0, out1 => "AI_PI3308_Truoc_Filter_HMI")
   END_RUNG
   // the same network as SCL:
   IF NOT "AI_HMI_Sim_Mode" THEN "AI_PI3308_Truoc_Filter_HMI" := 0.0; END_IF;
END_REGION

REGION Network 71: Reset AI_FT3309_Xa_Thanh_Pham_HMI về 0.0 khi ở chế độ chạy thật
   RUNG wire#powerrail
      I_Contact( "AI_HMI_Sim_Mode" )
      { S7_GenerateENO := "TRUE" } Move(in := 0.0, out1 => "AI_FT3309_Xa_Thanh_Pham_HMI")
   END_RUNG
   // the same network as SCL:
   IF NOT "AI_HMI_Sim_Mode" THEN "AI_FT3309_Xa_Thanh_Pham_HMI" := 0.0; END_IF;
END_REGION

REGION Network 72: Mô phỏng truyền thông Modbus TCP: Link Done nạp recipe PLC2 sang PLC1_HMI
   RUNG wire#powerrail
      Contact( "AI_HMI_Sim_Mode" )
      Contact( "AI_PLC1_Load_Default_Cmd" )
      Coil( "AI_PLC1_Load_Default_Done_Nhan_HMI" )
   END_RUNG
   // the same network as SCL:
   "AI_PLC1_Load_Default_Done_Nhan_HMI" := "AI_HMI_Sim_Mode" AND "AI_PLC1_Load_Default_Cmd";
END_REGION
END_FUNCTION

ORGANIZATION_BLOCK "OB30_PID_PLC1_Bon2"   // OB30, LAD, CyclicInterrupt
{ S7_Optimized_Access := 'TRUE' }
VERSION : 0.1
// stored: AutoNumber true, IsIECCheckEnabled false, SetENOAutomatically false
   VAR_INPUT
      Initial_Call : Bool;   // Initial call of this OB
      Event_Count : Int;   // Events discarded
   END_VAR
BEGIN

REGION Network 1: Initialize PID Bon 2 Kp parameter
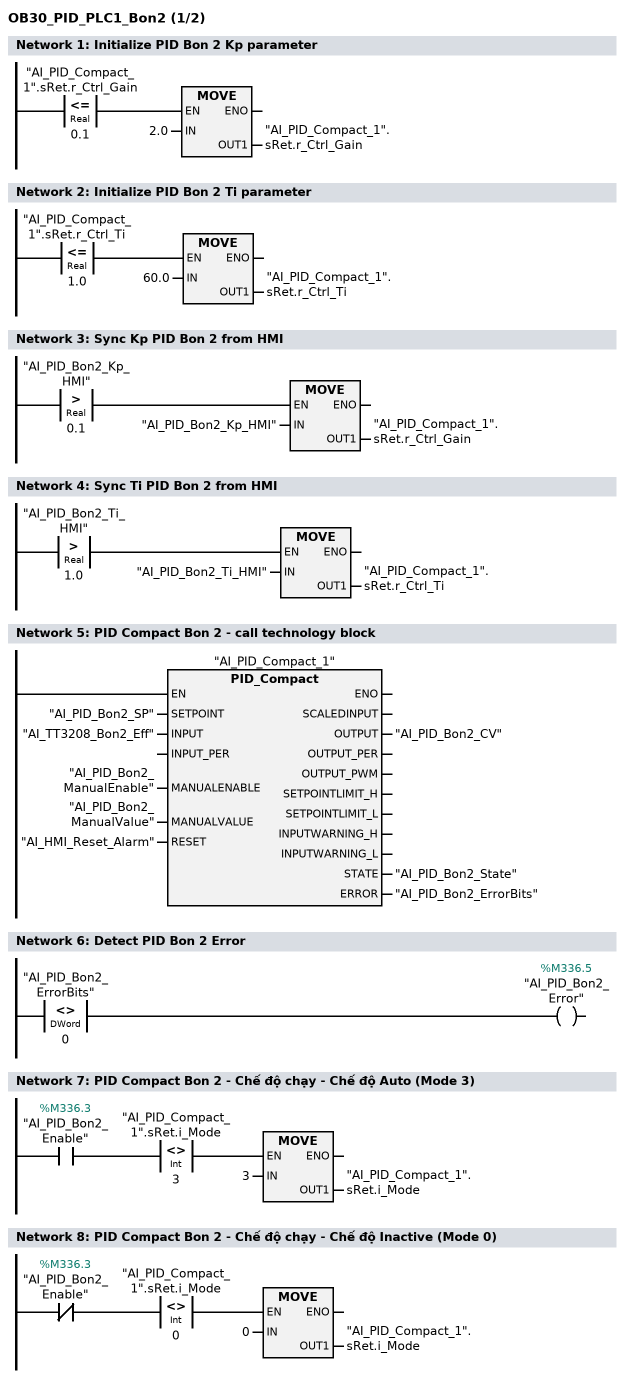
   RUNG wire#powerrail
      { S7_Templates := "SrcType := Real" } LE_Contact(in1 := "AI_PID_Compact_1".sRet.r_Ctrl_Gain, in2 := 0.1)
      { S7_GenerateENO := "TRUE" } Move(in := 2.0, out1 => "AI_PID_Compact_1".sRet.r_Ctrl_Gain)
   END_RUNG
   // the same network as SCL:
   IF "AI_PID_Compact_1".sRet.r_Ctrl_Gain <= 0.1 THEN "AI_PID_Compact_1".sRet.r_Ctrl_Gain := 2.0; END_IF;
END_REGION

REGION Network 2: Initialize PID Bon 2 Ti parameter
   RUNG wire#powerrail
      { S7_Templates := "SrcType := Real" } LE_Contact(in1 := "AI_PID_Compact_1".sRet.r_Ctrl_Ti, in2 := 1.0)
      { S7_GenerateENO := "TRUE" } Move(in := 60.0, out1 => "AI_PID_Compact_1".sRet.r_Ctrl_Ti)
   END_RUNG
   // the same network as SCL:
   IF "AI_PID_Compact_1".sRet.r_Ctrl_Ti <= 1.0 THEN "AI_PID_Compact_1".sRet.r_Ctrl_Ti := 60.0; END_IF;
END_REGION

REGION Network 3: Sync Kp PID Bon 2 from HMI
   RUNG wire#powerrail
      { S7_Templates := "SrcType := Real" } GT_Contact(in1 := "AI_PID_Bon2_Kp_HMI", in2 := 0.1)
      { S7_GenerateENO := "TRUE" } Move(in := "AI_PID_Bon2_Kp_HMI", out1 => "AI_PID_Compact_1".sRet.r_Ctrl_Gain)
   END_RUNG
   // the same network as SCL:
   IF "AI_PID_Bon2_Kp_HMI" > 0.1 THEN "AI_PID_Compact_1".sRet.r_Ctrl_Gain := "AI_PID_Bon2_Kp_HMI"; END_IF;
END_REGION

REGION Network 4: Sync Ti PID Bon 2 from HMI
   RUNG wire#powerrail
      { S7_Templates := "SrcType := Real" } GT_Contact(in1 := "AI_PID_Bon2_Ti_HMI", in2 := 1.0)
      { S7_GenerateENO := "TRUE" } Move(in := "AI_PID_Bon2_Ti_HMI", out1 => "AI_PID_Compact_1".sRet.r_Ctrl_Ti)
   END_RUNG
   // the same network as SCL:
   IF "AI_PID_Bon2_Ti_HMI" > 1.0 THEN "AI_PID_Compact_1".sRet.r_Ctrl_Ti := "AI_PID_Bon2_Ti_HMI"; END_IF;
END_REGION

REGION Network 5: PID Compact Bon 2 - call technology block
   RUNG wire#powerrail
      "AI_PID_Compact_1".PID_Compact(Setpoint := "AI_PID_Bon2_SP", Input := "AI_TT3208_Bon2_Eff", Input_PER :=, ManualEnable := "AI_PID_Bon2_ManualEnable", ManualValue := "AI_PID_Bon2_ManualValue", Reset := "AI_HMI_Reset_Alarm", ScaledInput =>, Output => "AI_PID_Bon2_CV", Output_PER =>, Output_PWM =>, SetpointLimit_H =>, SetpointLimit_L =>, InputWarning_H =>, InputWarning_L =>, State => "AI_PID_Bon2_State", Error => "AI_PID_Bon2_ErrorBits")
   END_RUNG
   // the same network as SCL:
   "AI_PID_Compact_1"(Setpoint := "AI_PID_Bon2_SP",   // PID_Compact
                      Input := "AI_TT3208_Bon2_Eff",
                      ManualEnable := "AI_PID_Bon2_ManualEnable",
                      ManualValue := "AI_PID_Bon2_ManualValue",
                      Reset := "AI_HMI_Reset_Alarm",
                      Output => "AI_PID_Bon2_CV",
                      State => "AI_PID_Bon2_State",
                      Error => "AI_PID_Bon2_ErrorBits");
END_REGION

REGION Network 6: Detect PID Bon 2 Error
   RUNG wire#powerrail
      { S7_Templates := "SrcType := DWord" } NE_Contact(in1 := "AI_PID_Bon2_ErrorBits", in2 := 0)
      Coil( "AI_PID_Bon2_Error" )
   END_RUNG
   // the same network as SCL:
   "AI_PID_Bon2_Error" := "AI_PID_Bon2_ErrorBits" <> 0;
END_REGION

REGION Network 7: PID Compact Bon 2 - Chế độ chạy - Chế độ Auto (Mode 3)
   RUNG wire#powerrail
      Contact( "AI_PID_Bon2_Enable" )
      { S7_Templates := "SrcType := Int" } NE_Contact(in1 := "AI_PID_Compact_1".sRet.i_Mode, in2 := 3)
      { S7_GenerateENO := "TRUE" } Move(in := 3, out1 => "AI_PID_Compact_1".sRet.i_Mode)
   END_RUNG
   // the same network as SCL:
   IF "AI_PID_Bon2_Enable" AND ("AI_PID_Compact_1".sRet.i_Mode <> 3) THEN
       "AI_PID_Compact_1".sRet.i_Mode := 3;
   END_IF;
END_REGION

REGION Network 8: PID Compact Bon 2 - Chế độ chạy - Chế độ Inactive (Mode 0)
   RUNG wire#powerrail
      I_Contact( "AI_PID_Bon2_Enable" )
      { S7_Templates := "SrcType := Int" } NE_Contact(in1 := "AI_PID_Compact_1".sRet.i_Mode, in2 := 0)
      { S7_GenerateENO := "TRUE" } Move(in := 0, out1 => "AI_PID_Compact_1".sRet.i_Mode)
   END_RUNG
   // the same network as SCL:
   IF NOT "AI_PID_Bon2_Enable" AND ("AI_PID_Compact_1".sRet.i_Mode <> 0) THEN
       "AI_PID_Compact_1".sRet.i_Mode := 0;
   END_IF;
END_REGION

REGION Network 9: Move PID Bon 2 CV to Steam Valve
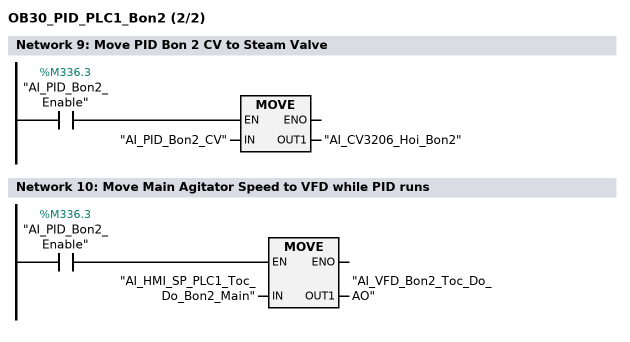
   RUNG wire#powerrail
      Contact( "AI_PID_Bon2_Enable" )
      { S7_GenerateENO := "TRUE" } Move(in := "AI_PID_Bon2_CV", out1 => "AI_CV3206_Hoi_Bon2")
   END_RUNG
   // the same network as SCL:
   IF "AI_PID_Bon2_Enable" THEN "AI_CV3206_Hoi_Bon2" := "AI_PID_Bon2_CV"; END_IF;
END_REGION

REGION Network 10: Move Main Agitator Speed to VFD while PID runs
   RUNG wire#powerrail
      Contact( "AI_PID_Bon2_Enable" )
      { S7_GenerateENO := "TRUE" } Move(in := "AI_HMI_SP_PLC1_Toc_Do_Bon2_Main", out1 => "AI_VFD_Bon2_Toc_Do_AO")
   END_RUNG
   // the same network as SCL:
   IF "AI_PID_Bon2_Enable" THEN "AI_VFD_Bon2_Toc_Do_AO" := "AI_HMI_SP_PLC1_Toc_Do_Bon2_Main"; END_IF;
END_REGION
END_ORGANIZATION_BLOCK

DATA_BLOCK "MB_CLIENT_DB"   // DB52
// stored: AutoNumber false, DBAccessibleFromOPCUA true, InstanceOfName MB_CLIENT, OfSystemLibElement MB_CLIENT, OfSystemLibVersion 3.1
"MB_CLIENT"
   // VAR_INPUT
   //    REQ : Bool;
   //    DISCONNECT : Bool;
   //    CONNECT_ID : UInt;
   //    IP_OCTET_1 : USInt;
   //    IP_OCTET_2 : USInt;
   //    IP_OCTET_3 : USInt;
   //    IP_OCTET_4 : USInt;
   //    IP_PORT : UInt;
   //    MB_MODE : USInt;
   //    MB_DATA_ADDR : UDInt;
   //    MB_DATA_LEN : UInt;
   // END_VAR
   // VAR_OUTPUT
   //    DONE : Bool;
   //    BUSY : Bool;
   //    ERROR : Bool;
   //    STATUS : Word;
   // END_VAR
   // VAR_IN_OUT
   //    MB_DATA_PTR : Variant;
   // END_VAR
   // VAR
   //    TCON_SFB { S7_SetPoint := 'True'} : TCON;
   //    TDISCON_SFB { S7_SetPoint := 'True'} : TDISCON;
   //    TSEND_SFB { S7_SetPoint := 'True'} : TSEND;
   //    TRCV_SFB { S7_SetPoint := 'True'} : TRCV;
   //    TCON_PARAM { S7_SetPoint := 'True'} : TCON_Param;
   //    PF_FREQUENCY : Real;
   //    BLOCKED_PROC_TIMEOUT : Real;
   //    RCV_TIMEOUT : Real;
   //    CURRENT_TIME_VALUE : DWord;
   //    SAVED_TIME_VALUE : DWord;
   //    XMT_TIME : DWord;
   //    SAVED_CONNECT_ID : Word;
   //    SAVED_IP_PORT : Word;
   //    SAVED_MODE : Byte;
   //    SAVED_IP1 : Byte;
   //    SAVED_IP2 : Byte;
   //    SAVED_IP3 : Byte;
   //    SAVED_IP4 : Byte;
   //    SAVED_DATA_ADDR : DWord;
   //    SAVED_DATA_LEN : Word;
   //    MB_STATE : Word;
   //    COMM_SENT_COUNT : Word;
   //    BYTE_COUNT : Word;
   //    BYTE_COUNTB : Byte;
   //    SAVED_START_ADDR : Word;
   //    MB_TRANSACTION_ID : Word;
   //    MB_UNIT_ID : Word;
   //    RETRIES : Word;
   //    INIT_OK : Bool;
   //    ACTIVE : Bool;
   //    CONNECTED : Bool;
   //    SAVED_MA_REQ : Bool;
   // END_VAR
BEGIN
   TCON_PARAM.CONNECTION_TYPE := 11;
   TCON_PARAM.LOCAL_DEVICE_ID := 64;
END_DATA_BLOCK

DATA_BLOCK "MB_COMM_LOAD_DB"   // DB50
// stored: AutoNumber false, DBAccessibleFromOPCUA true, InstanceOfName MB_COMM_LOAD, OfSystemLibElement MB_COMM_LOAD, OfSystemLibVersion 2.1
"MB_COMM_LOAD"
   // VAR_INPUT
   //    REQ : Bool;
   //    PORT : PORT;
   //    BAUD : UDInt;
   //    PARITY : UInt;
   //    FLOW_CTRL : UInt;
   //    RTS_ON_DLY : UInt;
   //    RTS_OFF_DLY : UInt;
   //    RESP_TO : UInt;
   // END_VAR
   // VAR_OUTPUT
   //    DONE : Bool;
   //    ERROR : Bool;
   //    STATUS : Word;
   // END_VAR
   // VAR_IN_OUT
   //    MB_DB : MB_BASE;
   // END_VAR
   // VAR
   //    ICHAR_GAP : UInt;
   //    RETRIES : UInt;
   //    WRREC_STATUS : Word;
   //    RDREC_STATUS : Word;
   //    SFC_STATUS : Word;
   //    Port_CFG_SFB : Array[0..25] of Byte;
   //    Send_CFG_SFB : Array[0..16] of Byte;
   //    Rcv_CFG_SFB : Array[0..60] of Byte;
   //    STOP_BITS : USInt;
   // END_VAR
BEGIN
END_DATA_BLOCK

DATA_BLOCK "MB_MASTER_DB"   // DB51
// stored: AutoNumber false, DBAccessibleFromOPCUA true, InstanceOfName MB_MASTER, OfSystemLibElement MB_MASTER, OfSystemLibVersion 2.2
"MB_MASTER"
   // // inherited from MB_BASE
   // VAR
   //    S_PORT : UInt;
   //    S_RESP_TO : UInt;
   //    S_ICHAR_GAP : UInt;
   //    S_RETRIES : UInt;
   // END_VAR
   // VAR_INPUT
   //    REQ : Bool;
   //    MB_ADDR : UInt;
   //    MODE : USInt;
   //    DATA_ADDR : UDInt;
   //    DATA_LEN : UInt;
   // END_VAR
   // VAR_OUTPUT
   //    DONE : Bool;
   //    BUSY : Bool;
   //    ERROR : Bool;
   //    STATUS : Word;
   // END_VAR
   // VAR_IN_OUT
   //    DATA_PTR : Variant;
   // END_VAR
   // VAR
   //    SEND_PTP_SFB : Array[0..11] of Byte;
   //    RCV_PTP_SFB : Array[0..11] of Byte;
   //    RCV_RST_SFB : Array[0..9] of Byte;
   //    PF_FREQUENCY : Real;
   //    BLOCKED_PROC_TIMEOUT : Real;
   //    CURRENT_TIME_VALUE : UDInt;
   //    SAVED_TIME_VALUE : UDInt;
   //    SAVED_SLAVE_ADDR : Word;
   //    SAVED_MODE : Word;
   //    SAVED_DATA_ADDR : DWord;
   //    SAVED_DATA_LEN : UInt;
   //    MB_STATE : UInt;
   //    COMM_SENT_COUNT : UInt;
   //    BYTE_COUNT : USInt;
   //    INIT_OK : Bool;
   //    ACTIVE : Bool;
   //    BROADCAST_FLAG : Bool;
   //    EXTENDED_ADDRESSING : Bool;
   //    SAVED_START_ADDR : UInt;
   //    TXBuf_Function_Offset : UDInt;
   //    TXBuf_Address_Offset : UDInt;
   //    TXBuf_Quantity_Offset : UDInt;
   // END_VAR
BEGIN
END_DATA_BLOCK
